Fanuc KAREL source: ko00088.KL

-- PROVISIONAL review KL for V770-1; original PC SHA256 fff7fa2fb2cb75166565dd8cb5c10e73cc48cc62f102afdb58e0a6badba44bd7
-- Incomplete behavior may be omitted. Consult companion uncertainty JSON. Do not deploy.
PROGRAM KO00088
%NOLOCKGROUP
BEGIN
  -- UNRESOLVED_PC offsets 5-12; opcodes 9D,23
  -- UNRESOLVED_PC offsets 17-69; opcodes 27,27,49,7E,AD,27,49,7E,AD,22,31,7E,4A
  -- UNRESOLVED_PC offsets 74-78; opcodes 7F
END KO00088
